Yaskawa INFORM job: NP_R2_D6-7(-90,0).JBI

/JOB
//NAME NP_R2_D6-7(-90,0)
//POS
///NPOS 226,226,226,7,0,0
///TOOL 0
///POSTYPE PULSE
///PULSE
C00000=-123771,-51516,-115725,-13623,87627,-38689
C00001=-121455,-23199,-59897,-13779,60370,-50624
C00002=-120980,-19231,-54009,-14327,58905,-50261
C00003=-120799,-17622,-51619,-14549,58311,-50114
C00004=-120556,-14660,-49400,-14696,58503,-50050
C00005=-120799,-17622,-51619,-14549,58311,-50114
C00006=-120577,-15061,-49748,-14680,58507,-50058
C00007=-120571,-15724,-48549,-14851,57463,-49911
C00008=-120577,-15061,-49748,-14680,58507,-50058
C00009=-120753,-16651,-52147,-14459,59117,-50206
C00010=-121212,-20561,-58050,-13917,60620,-50569
C00011=-121454,-23454,-59948,-13793,60273,-50611
C00012=-120979,-19473,-54057,-14342,58813,-50248
C00013=-120797,-17859,-51665,-14565,58220,-50101
C00014=-120553,-14896,-49449,-14711,58415,-50037
C00015=-120797,-17859,-51665,-14565,58220,-50101
C00016=-120579,-15306,-49796,-14693,58413,-50046
C00017=-120574,-15963,-48592,-14865,57370,-49898
C00018=-120579,-15306,-49796,-14693,58413,-50046
C00019=-120755,-16900,-52196,-14472,59021,-50194
C00020=-121216,-20823,-58102,-13928,60520,-50557
C00021=-106495,-23428,-61637,-28980,72363,-36797
C00022=-106812,-19463,-55754,-29056,70871,-36521
C00023=-106933,-17856,-53367,-29098,70268,-36407
C00024=-106931,-20142,-55044,-29122,70143,-36373
C00025=-106938,-17279,-54224,-28963,70990,-36599
C00026=-133546,-7733,-45466,-13794,64190,-44707
C00027=-133758,-9231,-47857,-13586,64840,-44859
C00028=-134310,-12890,-53732,-13070,66448,-45234
C00029=-123771,-51516,-115725,-13623,87627,-38689
C00030=-86075,-25351,-114548,-22023,103534,-46323
C00031=-1916,-99599,-106771,-38857,72414,-50929
C00032=-11939,-142274,-93704,-63886,60411,-60843
C00033=-145321,-153790,-109983,60060,49894,25240
C00034=-129666,-14096,-46483,37407,63914,42715
C00035=-126146,16315,-17987,38304,57375,41745
C00036=-121192,61832,37562,34472,60924,29272
C00037=-120892,68463,48193,35366,58208,28432
C00038=-120776,71410,52853,35802,57048,28051
C00039=-120618,75399,57628,36069,56255,27822
C00040=-120776,71410,52853,35802,57048,28051
C00041=-120647,74475,56479,35993,56457,27886
C00042=-120644,75009,58795,36441,55517,27519
C00043=-120647,74475,56479,35993,56457,27886
C00044=-120762,71390,51614,35521,57659,28289
C00045=-121056,64507,40605,34565,60456,29169
C00046=-120398,59747,38483,20798,46783,38557
C00047=-120671,66985,49589,22117,43945,37722
C00048=-120777,70199,54481,22743,42713,37337
C00049=-120618,74247,59313,22998,41843,37179
C00050=-120777,70199,54481,22743,42713,37337
C00051=-120648,73678,58595,22957,41989,37204
C00052=-120644,74357,61092,23480,40893,36890
C00053=-120648,73678,58595,22957,41989,37204
C00054=-120388,73947,60429,23187,41001,37063
C00055=-121271,74714,61360,23968,41090,36602
C00056=-120388,73947,60429,23187,41001,37063
C00057=-120279,70456,55149,22471,42318,37493
C00058=-120000,62716,43340,20999,45311,38405
C00059=-121723,64137,30756,2588,89456,-4741
C00060=-121476,68693,39450,2546,86443,-4721
C00061=-121380,70715,43187,2532,85180,-4714
C00062=-121215,74350,47517,2506,84379,-4675
C00063=-121380,70715,43187,2532,85180,-4714
C00064=-121251,73638,46632,2511,84559,-4683
C00065=-121248,73739,48411,2514,83516,-4703
C00066=-121251,73638,46632,2511,84559,-4683
C00067=-119687,70699,44873,2242,84086,-4167
C00068=-119611,72609,47141,2230,83669,-4148
C00069=-120492,73242,47903,2383,83551,-4447
C00070=-119611,72609,47141,2230,83669,-4148
C00071=-119687,70699,44873,2242,84086,-4167
C00072=-121380,70715,43187,2532,85180,-4714
C00073=-121476,68693,39450,2546,86443,-4721
C00074=-121723,64137,30756,2588,89456,-4741
C00075=-121195,62041,29551,4452,79876,-4663
C00076=-120896,67711,39055,4404,76933,-4667
C00077=-120779,70192,43147,4390,75688,-4671
C00078=-120621,73831,47473,4357,74889,-4645
C00079=-120779,70192,43147,4390,75688,-4671
C00080=-120643,72966,46413,4360,75097,-4646
C00081=-120639,73080,48209,4379,74053,-4682
C00082=-120643,72966,46413,4360,75097,-4646
C00083=-120757,70390,42181,4371,76381,-4639
C00084=-121052,64540,32403,4415,79399,-4632
C00085=-115157,36003,7988,23321,64834,29677
C00086=-115181,41156,16249,23796,62599,29181
C00087=-115190,43335,19713,24011,61672,28969
C00088=-115270,41020,17275,23984,61980,29006
C00089=-115193,43351,18486,23853,62374,29126
C00090=-126041,49576,26492,29186,64237,25134
C00091=-126129,47307,22864,28988,65205,25364
C00092=-126358,41979,14266,28570,67534,25895
C00093=-124388,42689,3738,9965,87004,-6391
C00094=-123783,46839,11122,9816,84556,-6388
C00095=-123548,48604,14206,9764,83551,-6389
C00096=-123551,48867,13240,9755,84271,-6334
C00097=-123706,46393,11818,9803,83898,-6414
C00098=-117782,45464,10780,8133,83426,-4498
C00099=-117970,43692,7714,8176,84412,-4495
C00100=-118453,39509,354,8297,86815,-4494
C00101=-120384,38102,11001,5107,57335,30164
C00102=-121079,43844,19421,5684,55160,29778
C00103=-121347,46260,22961,5922,54247,29619
C00104=-120874,45972,21710,5573,54832,29843
C00105=-121485,43938,20482,5987,54587,29582
C00106=-120018,45564,24177,5131,53056,30102
C00107=-119735,43114,20608,4887,53972,30263
C00108=-119004,37293,12129,4295,56151,30653
C00109=-126146,16315,-17987,38304,57375,41745
C00110=-129666,-14096,-46483,37407,63914,42715
C00111=-145321,-153790,-109983,60060,49894,25240
C00112=-118034,-154432,-110124,60042,49042,25380
C00113=-23634,-154432,-110124,60042,49042,25380
C00114=831,-150531,-109249,58084,47269,27129
C00115=-121136,-44216,-70470,-5914,46161,-46237
C00116=-120941,38078,2784,-5309,56330,-46754
C00117=-120196,62156,38269,-34294,60478,-29012
C00118=-120485,68900,49027,-35213,57744,-28163
C00119=-120597,71901,53753,-35664,56573,-27776
C00120=-120756,75925,58570,-35937,55772,-27545
C00121=-120597,71901,53753,-35664,56573,-27776
C00122=-120719,74995,57408,-35861,55982,-27608
C00123=-120715,75587,59796,-36326,55032,-27233
C00124=-120719,74995,57408,-35861,55982,-27608
C00125=-120608,71850,52469,-35375,57196,-28018
C00126=-120325,64848,41322,-34391,60013,-28908
C00127=-120971,61197,35744,-17694,55900,-31016
C00128=-120690,68057,46414,-18524,53064,-30387
C00129=-120582,71083,51078,-18909,51840,-30105
C00130=-120741,74997,55747,-19030,50986,-30009
C00131=-120582,71083,51078,-18909,51840,-30105
C00132=-120713,74340,54935,-19006,51146,-30028
C00133=-120709,74828,57190,-19310,50070,-29811
C00134=-120713,74340,54935,-19006,51146,-30028
C00135=-120998,74549,56692,-19085,50157,-29961
C00136=-120121,75289,57574,-19677,50211,-29569
C00137=-120998,74549,56692,-19085,50157,-29961
C00138=-121110,71284,51695,-18653,51457,-30267
C00139=-121397,63979,40406,-17738,54434,-30940
C00140=-119735,64258,30909,-2139,89051,4821
C00141=-119968,68871,39660,-2099,86032,4794
C00142=-120059,70919,43424,-2086,84767,4785
C00143=-120224,74561,47756,-2058,83968,4742
C00144=-120059,70919,43424,-2086,84767,4785
C00145=-120210,74155,47238,-2061,84079,4745
C00146=-120206,74290,49058,-2064,83029,4764
C00147=-120210,74155,47238,-2061,84079,4745
C00148=-121573,71362,45677,-1819,83572,4295
C00149=-121638,72966,47581,-1809,83223,4278
C00150=-120758,73614,48347,-1966,83106,4576
C00151=-121638,72966,47581,-1809,83223,4278
C00152=-121573,71362,45677,-1819,83572,4295
C00153=-120059,70919,43424,-2086,84767,4785
C00154=-119968,68871,39660,-2099,86032,4794
C00155=-119735,64258,30909,-2139,89051,4821
C00156=-120195,62467,30059,-4053,79421,4773
C00157=-120484,68208,39642,-4005,76466,4772
C00158=-120596,70723,43772,-3991,75214,4774
C00159=-120755,74380,48121,-3956,74412,4745
C00160=-120596,70723,43772,-3991,75214,4774
C00161=-120719,73521,47080,-3964,74612,4751
C00162=-120715,73671,48918,-3984,73560,4786
C00163=-120719,73521,47080,-3964,74612,4751
C00164=-120609,70909,42805,-3976,75903,4747
C00165=-120325,64982,32940,-4020,78935,4745
C00166=-120684,46164,21205,-28112,60266,-30898
C00167=-120683,46204,24154,-28601,58678,-30453
C00168=-120683,46271,25388,-28810,58038,-30270
C00169=-120686,46187,24054,-28585,58724,-30468
C00170=-120551,43918,22883,-28781,58376,-30309
C00171=-120683,46379,25414,-28799,58073,-30280
C00172=-120683,46314,24182,-28590,58713,-30463
C00173=-120684,46278,21237,-28101,60300,-30907
C00174=-120684,47343,12821,-8564,83099,5588
C00175=-120684,47348,12826,-8564,83098,5588
C00176=-120684,47350,12829,-8564,83098,5588
C00177=-120552,45134,10455,-8598,83431,5609
C00178=-120687,47604,11851,-8554,83823,5537
C00179=-120684,47293,12767,-8564,83107,5587
C00180=-120684,47291,12765,-8564,83107,5587
C00181=-120684,47286,12760,-8564,83108,5588
C00182=-120684,46249,18933,-4053,57953,-28008
C00183=-120684,46160,21215,-4118,56506,-27953
C00184=-120684,46157,22163,-4146,55923,-27930
C00185=-120551,43841,19698,-4212,56256,-27890
C00186=-121163,45883,20933,-3821,56514,-28142
C00187=-120683,46192,24181,-4206,54702,-27882
C00188=-120684,46156,23191,-4177,55291,-27905
C00189=-120684,46148,20806,-4107,56751,-27962
C00190=-120941,38078,2784,-5309,56330,-46754
C00191=-121025,6449,-31468,-5423,55852,-46694
C00192=-121119,-46995,-60266,-6864,38501,-45661
C00193=-56650,-90559,-87337,-45714,54134,-30117
C00194=3737,-1173,-65042,-31620,95650,-67595
C00195=-70607,2036,-67395,-11504,70170,-68245
C00196=-119853,-24034,-59175,14123,59074,50638
C00197=-120315,-19938,-53237,14680,57646,50274
C00198=-120491,-18280,-50826,14907,57065,50126
C00199=-120739,-15317,-48625,15056,57269,50060
C00200=-120491,-18280,-50826,14907,57065,50126
C00201=-120718,-15720,-48972,15039,57272,50069
C00202=-120712,-16317,-47726,15215,56233,49921
C00203=-120718,-15720,-48972,15039,57272,50069
C00204=-120547,-17358,-51390,14815,57869,50218
C00205=-120100,-21395,-57345,14263,59337,50583
C00206=-119855,-23768,-59136,14109,59184,50652
C00207=-120316,-19686,-53201,14665,57751,50288
C00208=-120493,-18032,-50791,14890,57167,50140
C00209=-120740,-15071,-48587,15039,57369,50074
C00210=-120493,-18032,-50791,14890,57167,50140
C00211=-120716,-15476,-48948,15020,57379,50085
C00212=-120711,-16079,-47707,15195,56340,49937
C00213=-120716,-15476,-48948,15020,57379,50085
C00214=-120546,-17109,-51366,14797,57978,50233
C00215=-120099,-21132,-57317,14246,59451,50598
C00216=-134824,-24307,-60893,29480,71143,36672
C00217=-134490,-20211,-54963,29562,69684,36403
C00218=-134363,-18554,-52558,29607,69092,36291
C00219=-134368,-18026,-53448,29466,69811,36483
C00220=-134362,-20842,-54222,29633,68959,36255
C00221=-107755,-8131,-44765,14075,63067,44728
C00222=-107547,-9673,-47176,13862,63706,44881
C00223=-107004,-13447,-53101,13337,65285,45258
C00224=-85700,1281,-76051,1309,91932,19786
C00225=-216,-87029,-95702,-46521,78496,-83300
BC00000=194152,749418,995208
BC00001=243652,746705,1075175
BC00002=243652,746705,1075175
BC00003=243652,746705,1075175
BC00004=243652,746705,1075175
BC00005=243652,746705,1075175
BC00006=243652,746705,1075175
BC00007=243652,746705,1075175
BC00008=243652,746705,1075175
BC00009=243652,746705,1075175
BC00010=243652,746705,1075175
BC00011=182506,757250,1075175
BC00012=182506,757250,1075175
BC00013=182506,757250,1075175
BC00014=182506,757250,1075175
BC00015=182506,757250,1075175
BC00016=182506,757250,1075175
BC00017=182506,757250,1075175
BC00018=182506,757250,1075175
BC00019=182506,757250,1075175
BC00020=182506,757250,1075175
BC00021=226486,761569,1075175
BC00022=226486,761569,1075175
BC00023=226486,761569,1075175
BC00024=226486,761569,1075175
BC00025=226486,761569,1075175
BC00026=226486,761569,1075175
BC00027=226486,761569,1075175
BC00028=226486,761569,1075175
BC00029=194152,749418,995208
BC00030=190434,735355,924438
BC00031=182227,704310,768212
BC00032=170902,666204,53
BC00033=170902,666204,53
BC00034=170902,666204,53
BC00035=170902,666204,53
BC00036=167884,674782,53
BC00037=167884,674782,53
BC00038=167884,674782,53
BC00039=167884,674782,53
BC00040=167884,674782,53
BC00041=167884,674782,53
BC00042=167884,674782,53
BC00043=167884,674782,53
BC00044=167884,674782,53
BC00045=167884,674782,53
BC00046=156929,666220,53
BC00047=156929,666220,53
BC00048=156929,666220,53
BC00049=156929,666220,53
BC00050=156929,666220,53
BC00051=156929,666220,53
BC00052=156929,666220,53
BC00053=156929,666220,53
BC00054=156929,666220,53
BC00055=156929,666220,53
BC00056=156929,666220,53
BC00057=156929,666220,53
BC00058=156929,666220,53
BC00059=165458,716793,64903
BC00060=165458,716793,64903
BC00061=165458,716793,64903
BC00062=165458,716793,64903
BC00063=165458,716793,64903
BC00064=165458,716793,64903
BC00065=165458,716793,64903
BC00066=165458,716793,64903
BC00067=165458,716793,64903
BC00068=165458,716793,64903
BC00069=165458,716793,64903
BC00070=165458,716793,64903
BC00071=165458,716793,64903
BC00072=165458,716793,64903
BC00073=165458,716793,64903
BC00074=165458,716793,64903
BC00075=146178,702943,44239
BC00076=146178,702943,44239
BC00077=146178,702943,44239
BC00078=146178,702943,44239
BC00079=146178,702943,44239
BC00080=146178,702943,44239
BC00081=146178,702943,44239
BC00082=146178,702943,44239
BC00083=146178,702943,44239
BC00084=146178,702943,44239
BC00085=156606,704627,53
BC00086=156606,704627,53
BC00087=156606,704627,53
BC00088=156606,704627,53
BC00089=156606,704627,53
BC00090=156606,704627,53
BC00091=156606,704627,53
BC00092=156606,704627,53
BC00093=144220,729084,3537
BC00094=144220,729084,3537
BC00095=144220,729084,3537
BC00096=144220,729084,3537
BC00097=144220,729084,3537
BC00098=144220,729084,3537
BC00099=144220,729084,3537
BC00100=144220,729084,3537
BC00101=173432,694880,53
BC00102=173432,694880,53
BC00103=173432,694880,53
BC00104=173432,694880,53
BC00105=173432,694880,53
BC00106=173432,694880,53
BC00107=173432,694880,53
BC00108=173432,694880,53
BC00109=170902,666204,53
BC00110=170902,666204,53
BC00111=170902,666204,53
BC00112=170902,666204,53
BC00113=170902,666204,53
BC00114=170902,666204,53
BC00115=268425,666204,53
BC00116=268425,666204,53
BC00117=270593,676138,53
BC00118=270593,676138,53
BC00119=270593,676138,53
BC00120=270593,676138,53
BC00121=270593,676138,53
BC00122=270593,676138,53
BC00123=270593,676138,53
BC00124=270593,676138,53
BC00125=270593,676138,53
BC00126=270593,676138,53
BC00127=281363,674163,53
BC00128=281363,674163,53
BC00129=281363,674163,53
BC00130=281363,674163,53
BC00131=281363,674163,53
BC00132=281363,674163,53
BC00133=281363,674163,53
BC00134=281363,674163,53
BC00135=281363,674163,53
BC00136=281363,674163,53
BC00137=281363,674163,53
BC00138=281363,674163,53
BC00139=281363,674163,53
BC00140=271621,717331,62121
BC00141=271621,717331,62121
BC00142=271621,717331,62121
BC00143=271621,717331,62121
BC00144=271621,717331,62121
BC00145=271621,717331,62121
BC00146=271621,717331,62121
BC00147=271621,717331,62121
BC00148=271621,717331,62121
BC00149=271621,717331,62121
BC00150=271621,717331,62121
BC00151=271621,717331,62121
BC00152=271621,717331,62121
BC00153=271621,717331,62121
BC00154=271621,717331,62121
BC00155=271621,717331,62121
BC00156=291354,703507,41702
BC00157=291354,703507,41702
BC00158=291354,703507,41702
BC00159=291354,703507,41702
BC00160=291354,703507,41702
BC00161=291354,703507,41702
BC00162=291354,703507,41702
BC00163=291354,703507,41702
BC00164=291354,703507,41702
BC00165=291354,703507,41702
BC00166=265943,691270,53
BC00167=265648,696742,53
BC00168=265530,698932,53
BC00169=265530,698932,53
BC00170=265530,698932,53
BC00171=300641,705051,53
BC00172=300759,702862,53
BC00173=301053,697389,53
BC00174=305010,723926,27777
BC00175=303349,729160,8919
BC00176=302685,731254,1375
BC00177=302685,731254,1375
BC00178=302685,731254,1375
BC00179=284050,728006,1066
BC00180=284714,725912,8610
BC00181=286374,720678,27469
BC00182=262622,690126,53
BC00183=264852,696041,53
BC00184=265744,698408,53
BC00185=265744,698408,53
BC00186=265744,698408,53
BC00187=261477,697681,53
BC00188=260585,695315,53
BC00189=258354,689399,53
BC00190=268425,666204,53
BC00191=268425,666204,53
BC00192=268425,666204,53
BC00193=228504,667032,174599
BC00194=26278,671229,1058787
BC00195=125651,715317,1068584
BC00196=192549,744724,1075175
BC00197=192549,744724,1075175
BC00198=192549,744724,1075175
BC00199=192549,744724,1075175
BC00200=192549,744724,1075175
BC00201=192549,744724,1075175
BC00202=192549,744724,1075175
BC00203=192549,744724,1075175
BC00204=192549,744724,1075175
BC00205=192549,744724,1075175
BC00206=253678,755374,1075175
BC00207=253678,755374,1075175
BC00208=253678,755374,1075175
BC00209=253678,755374,1075175
BC00210=253678,755374,1075175
BC00211=253678,755374,1075175
BC00212=253678,755374,1075175
BC00213=253678,755374,1075175
BC00214=253678,755374,1075175
BC00215=253678,755374,1075175
BC00216=209410,759520,1075175
BC00217=209410,759520,1075175
BC00218=209410,759520,1075175
BC00219=209410,759520,1075175
BC00220=209410,759520,1075175
BC00221=209410,759520,1075175
BC00222=209410,759520,1075175
BC00223=209410,759520,1075175
BC00224=180844,742474,1075175
BC00225=66580,674291,1075175
EC00000=-798156,0
EC00001=-798156,0
EC00002=-798156,0
EC00003=-798156,0
EC00004=-798156,0
EC00005=-798156,0
EC00006=-798156,0
EC00007=-798156,0
EC00008=-798156,0
EC00009=-798156,0
EC00010=-798156,0
EC00011=-798156,0
EC00012=-798156,0
EC00013=-798156,0
EC00014=-798156,0
EC00015=-798156,0
EC00016=-798156,0
EC00017=-798156,0
EC00018=-798156,0
EC00019=-798156,0
EC00020=-798156,0
EC00021=-798156,0
EC00022=-798156,0
EC00023=-798156,0
EC00024=-798156,0
EC00025=-798156,0
EC00026=-798156,0
EC00027=-798156,0
EC00028=-798156,0
EC00029=-798156,0
EC00030=-798156,0
EC00031=-798156,0
EC00032=-798156,0
EC00033=-798156,0
EC00034=-798156,0
EC00035=-798156,0
EC00036=-798156,0
EC00037=-798156,0
EC00038=-798156,0
EC00039=-798156,0
EC00040=-798156,0
EC00041=-798156,0
EC00042=-798156,0
EC00043=-798156,0
EC00044=-798156,0
EC00045=-798156,0
EC00046=-798156,0
EC00047=-798156,0
EC00048=-798156,0
EC00049=-798156,0
EC00050=-798156,0
EC00051=-798156,0
EC00052=-798156,0
EC00053=-798156,0
EC00054=-798156,0
EC00055=-798156,0
EC00056=-798156,0
EC00057=-798156,0
EC00058=-798156,0
EC00059=-798156,0
EC00060=-798156,0
EC00061=-798156,0
EC00062=-798156,0
EC00063=-798156,0
EC00064=-798156,0
EC00065=-798156,0
EC00066=-798156,0
EC00067=-798156,0
EC00068=-798156,0
EC00069=-798156,0
EC00070=-798156,0
EC00071=-798156,0
EC00072=-798156,0
EC00073=-798156,0
EC00074=-798156,0
EC00075=-798156,0
EC00076=-798156,0
EC00077=-798156,0
EC00078=-798156,0
EC00079=-798156,0
EC00080=-798156,0
EC00081=-798156,0
EC00082=-798156,0
EC00083=-798156,0
EC00084=-798156,0
EC00085=-798156,0
EC00086=-798156,0
EC00087=-798156,0
EC00088=-798156,0
EC00089=-798156,0
EC00090=-798156,0
EC00091=-798156,0
EC00092=-798156,0
EC00093=-798156,0
EC00094=-798156,0
EC00095=-798156,0
EC00096=-798156,0
EC00097=-798156,0
EC00098=-798156,0
EC00099=-798156,0
EC00100=-798156,0
EC00101=-798156,0
EC00102=-798156,0
EC00103=-798156,0
EC00104=-798156,0
EC00105=-798156,0
EC00106=-798156,0
EC00107=-798156,0
EC00108=-798156,0
EC00109=-798156,0
EC00110=-798156,0
EC00111=-798156,0
EC00112=-878342,206375
EC00113=-878342,851887
EC00114=-798156,1112951
EC00115=-798156,1112951
EC00116=-798156,1112951
EC00117=-798156,1112951
EC00118=-798156,1112951
EC00119=-798156,1112951
EC00120=-798156,1112951
EC00121=-798156,1112951
EC00122=-798156,1112951
EC00123=-798156,1112951
EC00124=-798156,1112951
EC00125=-798156,1112951
EC00126=-798156,1112951
EC00127=-798156,1112951
EC00128=-798156,1112951
EC00129=-798156,1112951
EC00130=-798156,1112951
EC00131=-798156,1112951
EC00132=-798156,1112951
EC00133=-798156,1112951
EC00134=-798156,1112951
EC00135=-798156,1112951
EC00136=-798156,1112951
EC00137=-798156,1112951
EC00138=-798156,1112951
EC00139=-798156,1112951
EC00140=-798156,1112951
EC00141=-798156,1112951
EC00142=-798156,1112951
EC00143=-798156,1112951
EC00144=-798156,1112951
EC00145=-798156,1112951
EC00146=-798156,1112951
EC00147=-798156,1112951
EC00148=-798156,1112951
EC00149=-798156,1112951
EC00150=-798156,1112951
EC00151=-798156,1112951
EC00152=-798156,1112951
EC00153=-798156,1112951
EC00154=-798156,1112951
EC00155=-798156,1112951
EC00156=-798156,1112951
EC00157=-798156,1112951
EC00158=-798156,1112951
EC00159=-798156,1112951
EC00160=-798156,1112951
EC00161=-798156,1112951
EC00162=-798156,1112951
EC00163=-798156,1112951
EC00164=-798156,1112951
EC00165=-798156,1112951
EC00166=-798156,1112951
EC00167=-798156,1112951
EC00168=-798156,1112951
EC00169=-798156,1112951
EC00170=-798156,1112951
EC00171=-798156,1112951
EC00172=-798156,1112951
EC00173=-798156,1112951
EC00174=-798156,1112951
EC00175=-798156,1112951
EC00176=-798156,1112951
EC00177=-798156,1112951
EC00178=-798156,1112951
EC00179=-798156,1112951
EC00180=-798156,1112951
EC00181=-798156,1112951
EC00182=-798156,1112951
EC00183=-798156,1112951
EC00184=-798156,1112951
EC00185=-798156,1112951
EC00186=-798156,1112951
EC00187=-798156,1112951
EC00188=-798156,1112951
EC00189=-798156,1112951
EC00190=-798156,1112951
EC00191=-798156,1112951
EC00192=-798156,1112951
EC00193=-798156,1112951
EC00194=-798156,1112951
EC00195=-798156,1112951
EC00196=-798156,1112951
EC00197=-798156,1112951
EC00198=-798156,1112951
EC00199=-798156,1112951
EC00200=-798156,1112951
EC00201=-798156,1112951
EC00202=-798156,1112951
EC00203=-798156,1112951
EC00204=-798156,1112951
EC00205=-798156,1112951
EC00206=-798156,1112951
EC00207=-798156,1112951
EC00208=-798156,1112951
EC00209=-798156,1112951
EC00210=-798156,1112951
EC00211=-798156,1112951
EC00212=-798156,1112951
EC00213=-798156,1112951
EC00214=-798156,1112951
EC00215=-798156,1112951
EC00216=-798156,1112951
EC00217=-798156,1112951
EC00218=-798156,1112951
EC00219=-798156,1112951
EC00220=-798156,1112951
EC00221=-798156,1112951
EC00222=-798156,1112951
EC00223=-798156,1112951
EC00224=-798156,1112951
EC00225=-798156,1112951
///POSTYPE BASE
///RECTAN
///RCONF 0,0,0,0,0,0,0,0,0,0,0,0,0,0,0,0,0,0,0,0,0,0,0,0
P00006=0.222,-3.123,-1.508,0.0000,0.0000,0.0000
P00021=-0.225,-6.128,-0.405,0.0000,0.0000,0.0000
P00022=0.222,-3.123,-1.508,0.0000,0.0000,0.0000
P00023=0.143,-0.036,0.682,0.0000,0.0000,0.0000
P00024=0.145,-0.552,1.326,0.0000,0.0000,0.0000
P00025=-2.003,0.006,0.728,0.0000,0.0000,0.0000
P00026=0.562,-0.002,-0.337,0.0000,0.0000,0.0000
//INST
///DATE 2024/02/03 16:15
///ATTR SC,RW
///GROUP1 RB1,BS1
///GROUP2 ST1
NOP
'Np_R2_D6-7(-90,0)
'Spoina W6
MOVJ C00000 BC00000 VJ=100.00  +MOVJ EC00000 VJ=100.00
'Path S3970
SSFTOF
MOVJ C00001 BC00001 VJ=100.00  +MOVJ EC00001 VJ=100.00
MOVL C00002 BC00002 V=400.0  +MOVJ EC00002 VJ=100.00
SMOVL C00003 BC00003 V=100.0  +MOVJ EC00003
SREFP 3 C00004 BC00004  +REFP EC00004
CALL JOB:SEARCH-R1-S1
SET P021 P006
SSFTON P021
SMOVL C00005 BC00005 V=100.0  +MOVJ EC00005
SMOVL C00006 BC00006 V=100.0  +MOVJ EC00006
SREFP 3 C00007 BC00007  +REFP EC00007
CALL JOB:SEARCH-R1-S1
SET P021 P006
SSFTON P021
SMOVL C00008 BC00008 V=100.0  +MOVJ EC00008
MOVL C00009 BC00009 V=400.0  +MOVJ EC00009 VJ=100.00
MOVL C00010 BC00010 V=1000.0  +MOVJ EC00010 VJ=100.00
'Path S3980
SSFTOF
MOVJ C00011 BC00011 VJ=100.00  +MOVJ EC00011 VJ=100.00
MOVL C00012 BC00012 V=400.0  +MOVJ EC00012 VJ=100.00
SMOVL C00013 BC00013 V=100.0  +MOVJ EC00013
SREFP 3 C00014 BC00014  +REFP EC00014
CALL JOB:SEARCH-R1-S1
SET P022 P006
SSFTON P022
SMOVL C00015 BC00015 V=100.0  +MOVJ EC00015
SMOVL C00016 BC00016 V=100.0  +MOVJ EC00016
SREFP 3 C00017 BC00017  +REFP EC00017
CALL JOB:SEARCH-R1-S1
SET P022 P006
SSFTON P022
SMOVL C00018 BC00018 V=100.0  +MOVJ EC00018
MOVL C00019 BC00019 V=400.0  +MOVJ EC00019 VJ=100.00
MOVL C00020 BC00020 V=1000.0  +MOVJ EC00020 VJ=100.00
'Path W3971
SSFTOF
SSFTON P021
MOVJ C00021 BC00021 VJ=100.00  +MOVJ EC00021 VJ=100.00
SMOVL C00022 BC00022 V=400.0  +MOVJ EC00022
SMOVL C00023 BC00023 V=150.0 PL=0  +MOVJ EC00023
SREFP 1 C00024 BC00024  +REFP EC00024
SREFP 2 C00025 BC00025  +REFP EC00025
MACRO1 MJ#(0) ARGF0
ARCON
SSFTON P022
SMOVL C00026 BC00026 V=10.0  +MOVJ EC00026
ARCOF
SMOVL C00027 BC00027 V=400.0  +MOVJ EC00027
SMOVL C00028 BC00028 V=1000.0  +MOVJ EC00028
SSFTOF
MOVJ C00029 BC00029 VJ=100.00  +MOVJ EC00029 VJ=100.00
MOVJ C00030 BC00030 VJ=100.00  +MOVJ EC00030 VJ=100.00
MOVJ C00031 BC00031 VJ=100.00  +MOVJ EC00031 VJ=100.00
MOVJ C00032 BC00032 VJ=100.00  +MOVJ EC00032 VJ=100.00
'wire_cut
'wire_cut
MOVJ C00033 BC00033 VJ=100.00  +MOVJ EC00033 VJ=100.00
MOVJ C00034 BC00034 VJ=100.00  +MOVJ EC00034 VJ=100.00
MOVJ C00035 BC00035 VJ=100.00  +MOVJ EC00035 VJ=100.00
'Path S3972
SSFTOF
MOVJ C00036 BC00036 VJ=100.00  +MOVJ EC00036 VJ=100.00
MOVL C00037 BC00037 V=400.0  +MOVJ EC00037 VJ=100.00
SMOVL C00038 BC00038 V=100.0  +MOVJ EC00038
SREFP 3 C00039 BC00039  +REFP EC00039
CALL JOB:SEARCH-R1-S1
SET P023 P006
SSFTON P023
SMOVL C00040 BC00040 V=100.0  +MOVJ EC00040
SMOVL C00041 BC00041 V=100.0  +MOVJ EC00041
SREFP 3 C00042 BC00042  +REFP EC00042
CALL JOB:SEARCH-R1-S1
SET P023 P006
SSFTON P023
SMOVL C00043 BC00043 V=100.0  +MOVJ EC00043
MOVL C00044 BC00044 V=400.0  +MOVJ EC00044 VJ=100.00
MOVL C00045 BC00045 V=1000.0  +MOVJ EC00045 VJ=100.00
'Path S3978
SSFTOF
MOVJ C00046 BC00046 VJ=100.00  +MOVJ EC00046 VJ=100.00
MOVL C00047 BC00047 V=400.0  +MOVJ EC00047 VJ=100.00
SMOVL C00048 BC00048 V=100.0  +MOVJ EC00048
SREFP 3 C00049 BC00049  +REFP EC00049
CALL JOB:SEARCH-R1-S1
SET P024 P006
SSFTON P024
SMOVL C00050 BC00050 V=100.0  +MOVJ EC00050
SMOVL C00051 BC00051 V=100.0  +MOVJ EC00051
SREFP 3 C00052 BC00052  +REFP EC00052
CALL JOB:SEARCH-R1-S1
SET P024 P006
SSFTON P024
SMOVL C00053 BC00053 V=100.0  +MOVJ EC00053
SMOVL C00054 BC00054 V=100.0  +MOVJ EC00054
SREFP 3 C00055 BC00055  +REFP EC00055
CALL JOB:SEARCH-R1-S1
SET P024 P006
SSFTON P024
SMOVL C00056 BC00056 V=100.0  +MOVJ EC00056
MOVL C00057 BC00057 V=400.0  +MOVJ EC00057 VJ=100.00
MOVL C00058 BC00058 V=1000.0  +MOVJ EC00058 VJ=100.00
'Path S3983
SSFTOF
MOVJ C00059 BC00059 VJ=100.00  +MOVJ EC00059 VJ=100.00
MOVL C00060 BC00060 V=400.0  +MOVJ EC00060 VJ=100.00
SMOVL C00061 BC00061 V=100.0  +MOVJ EC00061
SREFP 3 C00062 BC00062  +REFP EC00062
CALL JOB:SEARCH-R1-S1
SET P025 P006
SSFTON P025
SMOVL C00063 BC00063 V=100.0  +MOVJ EC00063
SMOVL C00064 BC00064 V=100.0  +MOVJ EC00064
SREFP 3 C00065 BC00065  +REFP EC00065
CALL JOB:SEARCH-R1-S1
SET P025 P006
SSFTON P025
SMOVL C00066 BC00066 V=100.0  +MOVJ EC00066
SMOVL C00067 BC00067 V=100.0  +MOVJ EC00067
SMOVL C00068 BC00068 V=100.0  +MOVJ EC00068
SREFP 3 C00069 BC00069  +REFP EC00069
CALL JOB:SEARCH-R1-S1
SET P025 P006
SSFTON P025
SMOVL C00070 BC00070 V=100.0  +MOVJ EC00070
SMOVL C00071 BC00071 V=100.0  +MOVJ EC00071
SMOVL C00072 BC00072 V=100.0  +MOVJ EC00072
MOVL C00073 BC00073 V=400.0  +MOVJ EC00073 VJ=100.00
MOVL C00074 BC00074 V=1000.0  +MOVJ EC00074 VJ=100.00
'Path S3979
SSFTOF
MOVJ C00075 BC00075 VJ=100.00  +MOVJ EC00075 VJ=100.00
MOVL C00076 BC00076 V=400.0  +MOVJ EC00076 VJ=100.00
SMOVL C00077 BC00077 V=100.0  +MOVJ EC00077
SREFP 3 C00078 BC00078  +REFP EC00078
CALL JOB:SEARCH-R1-S1
SET P026 P006
SSFTON P026
SMOVL C00079 BC00079 V=100.0  +MOVJ EC00079
SMOVL C00080 BC00080 V=100.0  +MOVJ EC00080
SREFP 3 C00081 BC00081  +REFP EC00081
CALL JOB:SEARCH-R1-S1
SET P026 P006
SSFTON P026
SMOVL C00082 BC00082 V=100.0  +MOVJ EC00082
MOVL C00083 BC00083 V=400.0  +MOVJ EC00083 VJ=100.00
MOVL C00084 BC00084 V=1000.0  +MOVJ EC00084 VJ=100.00
'Path W3973
SSFTOF
SSFTON P023
MOVJ C00085 BC00085 VJ=100.00  +MOVJ EC00085 VJ=100.00
SMOVL C00086 BC00086 V=400.0  +MOVJ EC00086
SMOVL C00087 BC00087 V=150.0 PL=0  +MOVJ EC00087
SREFP 1 C00088 BC00088  +REFP EC00088
SREFP 2 C00089 BC00089  +REFP EC00089
MACRO1 MJ#(0) ARGF0
ARCON
SSFTON P024
SMOVL C00090 BC00090 V=10.0  +MOVJ EC00090
ARCOF
SMOVL C00091 BC00091 V=400.0  +MOVJ EC00091
SMOVL C00092 BC00092 V=1000.0  +MOVJ EC00092
SSFTOF
'Path W3981
SSFTOF
SSFTON P026
MOVJ C00093 BC00093 VJ=100.00  +MOVJ EC00093 VJ=100.00
SMOVL C00094 BC00094 V=400.0  +MOVJ EC00094
SMOVL C00095 BC00095 V=150.0 PL=0  +MOVJ EC00095
SREFP 1 C00096 BC00096  +REFP EC00096
SREFP 2 C00097 BC00097  +REFP EC00097
MACRO1 MJ#(0) ARGF0
ARCON
SSFTON P025
SMOVL C00098 BC00098 V=10.0  +MOVJ EC00098
ARCOF
SMOVL C00099 BC00099 V=400.0  +MOVJ EC00099
SMOVL C00100 BC00100 V=1000.0  +MOVJ EC00100
SSFTOF
'Path W3982
SSFTOF
SSFTON P025
MOVJ C00101 BC00101 VJ=100.00  +MOVJ EC00101 VJ=100.00
SMOVL C00102 BC00102 V=400.0  +MOVJ EC00102
SMOVL C00103 BC00103 V=150.0 PL=0  +MOVJ EC00103
SREFP 1 C00104 BC00104  +REFP EC00104
SREFP 2 C00105 BC00105  +REFP EC00105
MACRO1 MJ#(0) ARGF0
ARCON
SSFTON P024
SMOVL C00106 BC00106 V=10.0  +MOVJ EC00106
ARCOF
SMOVL C00107 BC00107 V=400.0  +MOVJ EC00107
SMOVL C00108 BC00108 V=1000.0  +MOVJ EC00108
SSFTOF
MOVJ C00109 BC00109 VJ=100.00  +MOVJ EC00109 VJ=100.00
MOVJ C00110 BC00110 VJ=100.00  +MOVJ EC00110 VJ=100.00
MOVJ C00111 BC00111 VJ=100.00  +MOVJ EC00111 VJ=100.00
MOVJ C00112 BC00112 VJ=100.00  +MOVJ EC00112 VJ=100.00
MOVJ C00113 BC00113 VJ=100.00  +MOVJ EC00113 VJ=100.00
MOVJ C00114 BC00114 VJ=100.00  +MOVJ EC00114 VJ=100.00
'wire_cut
'wire_cut
MOVJ C00115 BC00115 VJ=100.00  +MOVJ EC00115 VJ=100.00
MOVJ C00116 BC00116 VJ=100.00  +MOVJ EC00116 VJ=100.00
'wire_cut
'Spoina W7
'Path S3987
SSFTOF
MOVJ C00117 BC00117 VJ=100.00  +MOVJ EC00117 VJ=100.00
MOVL C00118 BC00118 V=400.0  +MOVJ EC00118 VJ=100.00
SMOVL C00119 BC00119 V=100.0  +MOVJ EC00119
SREFP 3 C00120 BC00120  +REFP EC00120
CALL JOB:SEARCH-R1-S1
SET P023 P006
SSFTON P023
SMOVL C00121 BC00121 V=100.0  +MOVJ EC00121
SMOVL C00122 BC00122 V=100.0  +MOVJ EC00122
SREFP 3 C00123 BC00123  +REFP EC00123
CALL JOB:SEARCH-R1-S1
SET P023 P006
SSFTON P023
SMOVL C00124 BC00124 V=100.0  +MOVJ EC00124
MOVL C00125 BC00125 V=400.0  +MOVJ EC00125 VJ=100.00
MOVL C00126 BC00126 V=1000.0  +MOVJ EC00126 VJ=100.00
'Path S3988
SSFTOF
MOVJ C00127 BC00127 VJ=100.00  +MOVJ EC00127 VJ=100.00
MOVL C00128 BC00128 V=400.0  +MOVJ EC00128 VJ=100.00
SMOVL C00129 BC00129 V=100.0  +MOVJ EC00129
SREFP 3 C00130 BC00130  +REFP EC00130
CALL JOB:SEARCH-R1-S1
SET P024 P006
SSFTON P024
SMOVL C00131 BC00131 V=100.0  +MOVJ EC00131
SMOVL C00132 BC00132 V=100.0  +MOVJ EC00132
SREFP 3 C00133 BC00133  +REFP EC00133
CALL JOB:SEARCH-R1-S1
SET P024 P006
SSFTON P024
SMOVL C00134 BC00134 V=100.0  +MOVJ EC00134
SMOVL C00135 BC00135 V=100.0  +MOVJ EC00135
SREFP 3 C00136 BC00136  +REFP EC00136
CALL JOB:SEARCH-R1-S1
SET P024 P006
SSFTON P024
SMOVL C00137 BC00137 V=100.0  +MOVJ EC00137
MOVL C00138 BC00138 V=400.0  +MOVJ EC00138 VJ=100.00
MOVL C00139 BC00139 V=1000.0  +MOVJ EC00139 VJ=100.00
'Path S3989
SSFTOF
MOVJ C00140 BC00140 VJ=100.00  +MOVJ EC00140 VJ=100.00
MOVL C00141 BC00141 V=400.0  +MOVJ EC00141 VJ=100.00
SMOVL C00142 BC00142 V=100.0  +MOVJ EC00142
SREFP 3 C00143 BC00143  +REFP EC00143
CALL JOB:SEARCH-R1-S1
SET P025 P006
SSFTON P025
SMOVL C00144 BC00144 V=100.0  +MOVJ EC00144
SMOVL C00145 BC00145 V=100.0  +MOVJ EC00145
SREFP 3 C00146 BC00146  +REFP EC00146
CALL JOB:SEARCH-R1-S1
SET P025 P006
SSFTON P025
SMOVL C00147 BC00147 V=100.0  +MOVJ EC00147
SMOVL C00148 BC00148 V=100.0  +MOVJ EC00148
SMOVL C00149 BC00149 V=100.0  +MOVJ EC00149
SREFP 3 C00150 BC00150  +REFP EC00150
CALL JOB:SEARCH-R1-S1
SET P025 P006
SSFTON P025
SMOVL C00151 BC00151 V=100.0  +MOVJ EC00151
SMOVL C00152 BC00152 V=100.0  +MOVJ EC00152
SMOVL C00153 BC00153 V=100.0  +MOVJ EC00153
MOVL C00154 BC00154 V=400.0  +MOVJ EC00154 VJ=100.00
MOVL C00155 BC00155 V=1000.0  +MOVJ EC00155 VJ=100.00
'Path S3990
SSFTOF
MOVJ C00156 BC00156 VJ=100.00  +MOVJ EC00156 VJ=100.00
MOVL C00157 BC00157 V=400.0  +MOVJ EC00157 VJ=100.00
SMOVL C00158 BC00158 V=100.0  +MOVJ EC00158
SREFP 3 C00159 BC00159  +REFP EC00159
CALL JOB:SEARCH-R1-S1
SET P026 P006
SSFTON P026
SMOVL C00160 BC00160 V=100.0  +MOVJ EC00160
SMOVL C00161 BC00161 V=100.0  +MOVJ EC00161
SREFP 3 C00162 BC00162  +REFP EC00162
CALL JOB:SEARCH-R1-S1
SET P026 P006
SSFTON P026
SMOVL C00163 BC00163 V=100.0  +MOVJ EC00163
MOVL C00164 BC00164 V=400.0  +MOVJ EC00164 VJ=100.00
MOVL C00165 BC00165 V=1000.0  +MOVJ EC00165 VJ=100.00
'Path W3991
SSFTOF
SSFTON P023
MOVJ C00166 BC00166 VJ=100.00  +MOVJ EC00166 VJ=100.00
SMOVL C00167 BC00167 V=400.0  +MOVJ EC00167
SMOVL C00168 BC00168 V=150.0 PL=0  +MOVJ EC00168
SREFP 1 C00169 BC00169  +REFP EC00169
SREFP 2 C00170 BC00170  +REFP EC00170
MACRO1 MJ#(0) ARGF0
ARCON
SSFTON P024
SMOVL C00171 BC00171 V=10.0  +MOVJ EC00171
ARCOF
SMOVL C00172 BC00172 V=400.0  +MOVJ EC00172
SMOVL C00173 BC00173 V=1000.0  +MOVJ EC00173
SSFTOF
'Path W3992
SSFTOF
SSFTON P026
MOVJ C00174 BC00174 VJ=100.00  +MOVJ EC00174 VJ=100.00
SMOVL C00175 BC00175 V=400.0  +MOVJ EC00175
SMOVL C00176 BC00176 V=150.0 PL=0  +MOVJ EC00176
SREFP 1 C00177 BC00177  +REFP EC00177
SREFP 2 C00178 BC00178  +REFP EC00178
MACRO1 MJ#(0) ARGF0
ARCON
SSFTON P025
SMOVL C00179 BC00179 V=10.0  +MOVJ EC00179
ARCOF
SMOVL C00180 BC00180 V=400.0  +MOVJ EC00180
SMOVL C00181 BC00181 V=1000.0  +MOVJ EC00181
SSFTOF
'Path W3993
SSFTOF
SSFTON P025
MOVJ C00182 BC00182 VJ=100.00  +MOVJ EC00182 VJ=100.00
SMOVL C00183 BC00183 V=400.0  +MOVJ EC00183
SMOVL C00184 BC00184 V=150.0 PL=0  +MOVJ EC00184
SREFP 1 C00185 BC00185  +REFP EC00185
SREFP 2 C00186 BC00186  +REFP EC00186
MACRO1 MJ#(0) ARGF0
ARCON
SSFTON P024
SMOVL C00187 BC00187 V=10.0  +MOVJ EC00187
ARCOF
SMOVL C00188 BC00188 V=400.0  +MOVJ EC00188
SMOVL C00189 BC00189 V=1000.0  +MOVJ EC00189
SSFTOF
'wire_cut
MOVJ C00190 BC00190 VJ=100.00  +MOVJ EC00190 VJ=100.00
MOVJ C00191 BC00191 VJ=100.00  +MOVJ EC00191 VJ=100.00
MOVJ C00192 BC00192 VJ=100.00  +MOVJ EC00192 VJ=100.00
MOVJ C00193 BC00193 VJ=10.00  +MOVJ EC00193 VJ=10.00
MOVJ C00194 BC00194 VJ=100.00  +MOVJ EC00194 VJ=100.00
MOVJ C00195 BC00195 VJ=100.00  +MOVJ EC00195 VJ=100.00
'Path S3984
SSFTOF
MOVJ C00196 BC00196 VJ=100.00  +MOVJ EC00196 VJ=100.00
MOVL C00197 BC00197 V=400.0  +MOVJ EC00197 VJ=100.00
SMOVL C00198 BC00198 V=100.0  +MOVJ EC00198
SREFP 3 C00199 BC00199  +REFP EC00199
CALL JOB:SEARCH-R1-S1
SET P021 P006
SSFTON P021
SMOVL C00200 BC00200 V=100.0  +MOVJ EC00200
SMOVL C00201 BC00201 V=100.0  +MOVJ EC00201
SREFP 3 C00202 BC00202  +REFP EC00202
CALL JOB:SEARCH-R1-S1
SET P021 P006
SSFTON P021
SMOVL C00203 BC00203 V=100.0  +MOVJ EC00203
MOVL C00204 BC00204 V=400.0  +MOVJ EC00204 VJ=100.00
MOVL C00205 BC00205 V=1000.0  +MOVJ EC00205 VJ=100.00
'Path S3985
SSFTOF
MOVJ C00206 BC00206 VJ=100.00  +MOVJ EC00206 VJ=100.00
MOVL C00207 BC00207 V=400.0  +MOVJ EC00207 VJ=100.00
SMOVL C00208 BC00208 V=100.0  +MOVJ EC00208
SREFP 3 C00209 BC00209  +REFP EC00209
CALL JOB:SEARCH-R1-S1
SET P022 P006
SSFTON P022
SMOVL C00210 BC00210 V=100.0  +MOVJ EC00210
SMOVL C00211 BC00211 V=100.0  +MOVJ EC00211
SREFP 3 C00212 BC00212  +REFP EC00212
CALL JOB:SEARCH-R1-S1
SET P022 P006
SSFTON P022
SMOVL C00213 BC00213 V=100.0  +MOVJ EC00213
MOVL C00214 BC00214 V=400.0  +MOVJ EC00214 VJ=100.00
MOVL C00215 BC00215 V=1000.0  +MOVJ EC00215 VJ=100.00
'Path W3986
SSFTOF
SSFTON P021
MOVJ C00216 BC00216 VJ=100.00  +MOVJ EC00216 VJ=100.00
SMOVL C00217 BC00217 V=400.0  +MOVJ EC00217
SMOVL C00218 BC00218 V=150.0 PL=0  +MOVJ EC00218
SREFP 1 C00219 BC00219  +REFP EC00219
SREFP 2 C00220 BC00220  +REFP EC00220
MACRO1 MJ#(0) ARGF0
ARCON
SSFTON P022
SMOVL C00221 BC00221 V=10.0  +MOVJ EC00221
ARCOF
SMOVL C00222 BC00222 V=400.0  +MOVJ EC00222
SMOVL C00223 BC00223 V=1000.0  +MOVJ EC00223
SSFTOF
MOVJ C00224 BC00224 VJ=100.00  +MOVJ EC00224 VJ=100.00
MOVJ C00225 BC00225 VJ=100.00  +MOVJ EC00225 VJ=100.00
END
